FUNCTION_BLOCK Randomizer
VAR
  _rndUniform : RandomUniform(seed:=0, lowerBound:=0, upperBound:=1);
  _rnd : IRandom;
END_VAR

METHOD FB_init : BOOL
VAR_INPUT
	bInitRetains : BOOL; // if TRUE, the retain variables are initialized (warm start / cold start)
	bInCopyCode : BOOL;  // if TRUE, the instance afterwards gets moved into the copy code (online change)
  rnd : IRandom;
END_VAR
_rnd := rnd;
END_METHOD

METHOD Fill
VAR_INPUT
  data : POINTER TO LREAL;
  size : INT;
END_VAR
VAR
  i : INT;
END_VAR
FOR i:=0 TO size-1
DO
  data[i] := _rnd.Next();
END_FOR
END_METHOD

METHOD FillMax
VAR_INPUT
  data : POINTER TO LREAL;
  size : INT;
  offset : POINTER TO LREAL;
END_VAR
VAR
  i : INT;
END_VAR
FOR i:=0 TO size-1
DO
  data[i] := _rnd.Next() + ABS(offset[i]);
END_FOR
END_METHOD

METHOD FillMin
VAR_INPUT
  data : POINTER TO LREAL;
  size : INT;
  offset : POINTER TO LREAL;
END_VAR
VAR
  i : INT;
END_VAR
FOR i:=0 TO size-1
DO
  data[i] := _rnd.Next() - ABS(offset[i]);
END_FOR
END_METHOD

METHOD FillOrZero
VAR_INPUT
  data : POINTER TO LREAL;
  size : INT;
  p : LREAL; // value between 0-1 to adjust the probability of "fill with random number" to "fill with zero". p = 0.9 means that 10% of values are filled with zero
END_VAR
VAR
  i : INT;
END_VAR
FOR i:=0 TO size-1
DO
  data[i] := SEL(_rndUniform.Next() < p, 0, _rnd.Next());
END_FOR
END_METHOD

END_FUNCTION_BLOCK

(* stored: Version 1.1.0.1, ProductVersion 3.1.4024.9
   POU Randomizer: Id {bab5e9c4-5a1f-4e70-8b4d-c4488a914d49}, SpecialFunc None
   Method FB_init: Id {4c3db243-9a05-4916-8518-95991e110a2a}
   Method Fill: Id {dfb58af6-4571-40c0-92e3-c2c910cd566d}
   Method FillMax: Id {c6eb80dc-521b-4003-9dde-700ce36a116b}
   Method FillMin: Id {a97d6307-80ff-438f-a50a-defe7e4f4db5}
   Method FillOrZero: Id {138d4024-11cf-4a39-8b3f-1585955de9a9} *)
